FUNCTION_BLOCK FB_HYDRAULIC_VALVE
VAR_INPUT
END_VAR
VAR_OUTPUT
	SolenoidExtend	: BOOL;
	SolenoidRetract	: BOOL;
END_VAR
VAR
END_VAR

METHOD Extend : BOOL
VAR_INPUT
END_VAR
SolenoidExtend := TRUE;
SolenoidRetract := FALSE;
END_METHOD

METHOD Neutral : BOOL
VAR_INPUT
END_VAR
SolenoidExtend := FALSE;
SolenoidRetract := FALSE;
END_METHOD

METHOD Retract : BOOL
VAR_INPUT
END_VAR
SolenoidExtend := FALSE;
SolenoidRetract := TRUE;
END_METHOD

END_FUNCTION_BLOCK

(* stored: Version 1.1.0.1, ProductVersion 3.1.4024.12
   POU FB_HYDRAULIC_VALVE: Id {b136142e-429b-4c48-853b-9aa6b2b9c920}, SpecialFunc None
   Method Extend: Id {376c3008-aa6a-4c72-a032-f4909481f840}
   Method Neutral: Id {5e107f79-66ac-44f3-b152-d0bd24930a39}
   Method Retract: Id {d684bcf7-76cd-46c9-aa2e-ea5057b17140} *)
